// TIA Portal V21 export
VAR_GLOBAL   // PLC tag table "K_TipoSendRecive"
END_VAR
VAR_GLOBAL CONSTANT   // user constants
   K_TipoSendRecive_Send : Int := 0;
   K_TipoSendRecive_Receive : Int := 1;
END_VAR
